Fanuc TP program (LS listing): SET_LOAD_PR.LS

/PROG  SET_LOAD_PR
/ATTR
OWNER		= MNEDITOR;
COMMENT		= "Set Grinder Load";
PROG_SIZE	= 3133;
CREATE		= DATE 28-11-03  TIME 05:11:18;
MODIFIED	= DATE 31-06-20  TIME 05:46:50;
FILE_NAME	= SET_SLOT;
VERSION		= 0;
LINE_COUNT	= 179;
MEMORY_SIZE	= 3693;
PROTECT		= READ_WRITE;
TCD:  STACK_SIZE	= 0,
      TASK_PRIORITY	= 50,
      TIME_SLICE	= 0,
      BUSY_LAMP_OFF	= 0,
      ABORT_REQUEST	= 0,
      PAUSE_REQUEST	= 0;
DEFAULT_GROUP	= *,*,*,*,*;
CONTROL_CODE	= 00000000 00000000;
/APPL
/APPL

AUTO_SINGULARITY_HEADER;
  ENABLE_SINGULARITY_AVOIDANCE   : TRUE;
/MN
   1:  JMP LBL[1] ;
   2:  !******************************* ;
   3:  !COMPANY ;
   4:  !PROJECT 0000000 ;
   5:  !CUSTOMER Example Cell ;
   6:  ! ;
   7:  !Date: March 24, 2022 ;
   8:  ! ;
   9:  !This program calculates the part ;
  10:  !tray LD position offsets. ;
  11:  ! ;
  12:  !******************************* ;
  13:  LBL[1:Begin] ;
  14:  !******************************* ;
  15:   ;
  16:  R[51:Part Style]=GI[3:Style Code]    ;
  17:   ;
  18:  !******************************* ;
  19:  LBL[5:Set Z values] ;
  20:  !******************************* ;
  21:   ;
  22:  SELECT R[51:Part Style]=1,JMP LBL[101] ;
  23:         =2,JMP LBL[102] ;
  24:         =3,JMP LBL[103] ;
  25:         =4,JMP LBL[104] ;
  26:         =5,JMP LBL[105] ;
  27:         =6,JMP LBL[106] ;
  28:         =7,JMP LBL[107] ;
  29:         =8,JMP LBL[108] ;
  30:         =9,JMP LBL[109] ;
  31:         =10,JMP LBL[110] ;
  32:         =11,JMP LBL[111] ;
  33:         =12,JMP LBL[112] ;
  34:         =13,JMP LBL[113] ;
  35:         =14,JMP LBL[114] ;
  36:         =15,JMP LBL[115] ;
  37:         =16,JMP LBL[116] ;
  38:         =17,JMP LBL[117] ;
  39:         =18,JMP LBL[118] ;
  40:         =19,JMP LBL[119] ;
  41:         =20,JMP LBL[120] ;
  42:         =21,JMP LBL[121] ;
  43:         =22,JMP LBL[122] ;
  44:         ELSE,JMP LBL[900] ;
  45:   ;
  46:  LBL[101] ;
  47:  R[56:Grinder Ld PR]=121    ;
  48:  R[57:Grinder Unld PR]=131    ;
  49:  R[58:Audit Ld PR]=151    ;
  50:  JMP LBL[200] ;
  51:   ;
  52:  LBL[102] ;
  53:  R[56:Grinder Ld PR]=122    ;
  54:  R[57:Grinder Unld PR]=132    ;
  55:  R[58:Audit Ld PR]=152    ;
  56:  JMP LBL[200] ;
  57:   ;
  58:  LBL[103] ;
  59:  R[56:Grinder Ld PR]=123    ;
  60:  R[57:Grinder Unld PR]=133    ;
  61:  R[58:Audit Ld PR]=153    ;
  62:  JMP LBL[200] ;
  63:   ;
  64:  LBL[104] ;
  65:  R[56:Grinder Ld PR]=124    ;
  66:  R[57:Grinder Unld PR]=134    ;
  67:  R[58:Audit Ld PR]=154    ;
  68:  JMP LBL[200] ;
  69:   ;
  70:  LBL[105] ;
  71:  R[56:Grinder Ld PR]=125    ;
  72:  R[57:Grinder Unld PR]=135    ;
  73:  R[58:Audit Ld PR]=155    ;
  74:  JMP LBL[200] ;
  75:   ;
  76:  LBL[106] ;
  77:  R[56:Grinder Ld PR]=126    ;
  78:  R[57:Grinder Unld PR]=136    ;
  79:  R[58:Audit Ld PR]=156    ;
  80:  JMP LBL[200] ;
  81:   ;
  82:  LBL[107] ;
  83:  R[56:Grinder Ld PR]=127    ;
  84:  R[57:Grinder Unld PR]=137    ;
  85:  R[58:Audit Ld PR]=157    ;
  86:  JMP LBL[200] ;
  87:   ;
  88:  LBL[108] ;
  89:  R[56:Grinder Ld PR]=128    ;
  90:  R[57:Grinder Unld PR]=138    ;
  91:  R[58:Audit Ld PR]=158    ;
  92:  JMP LBL[200] ;
  93:   ;
  94:  LBL[109] ;
  95:  R[56:Grinder Ld PR]=129    ;
  96:  R[57:Grinder Unld PR]=139    ;
  97:  R[58:Audit Ld PR]=159    ;
  98:  JMP LBL[200] ;
  99:   ;
 100:  LBL[110] ;
 101:  R[56:Grinder Ld PR]=130    ;
 102:  R[57:Grinder Unld PR]=140    ;
 103:  R[58:Audit Ld PR]=160    ;
 104:  JMP LBL[200] ;
 105:   ;
 106:  LBL[111] ;
 107:  R[56:Grinder Ld PR]=201    ;
 108:  R[57:Grinder Unld PR]=141    ;
 109:  JMP LBL[200] ;
 110:   ;
 111:  LBL[112] ;
 112:  R[56:Grinder Ld PR]=202    ;
 113:  R[57:Grinder Unld PR]=142    ;
 114:  JMP LBL[200] ;
 115:   ;
 116:  LBL[113] ;
 117:  R[56:Grinder Ld PR]=203    ;
 118:  R[57:Grinder Unld PR]=143    ;
 119:  JMP LBL[200] ;
 120:   ;
 121:  LBL[114] ;
 122:  R[56:Grinder Ld PR]=204    ;
 123:  R[57:Grinder Unld PR]=144    ;
 124:  JMP LBL[200] ;
 125:   ;
 126:  LBL[115] ;
 127:  R[56:Grinder Ld PR]=205    ;
 128:  R[57:Grinder Unld PR]=145    ;
 129:  JMP LBL[200] ;
 130:   ;
 131:  LBL[116] ;
 132:  R[56:Grinder Ld PR]=206    ;
 133:  R[57:Grinder Unld PR]=146    ;
 134:  JMP LBL[200] ;
 135:   ;
 136:  LBL[117] ;
 137:  R[56:Grinder Ld PR]=207    ;
 138:  R[57:Grinder Unld PR]=147    ;
 139:  JMP LBL[200] ;
 140:   ;
 141:  LBL[118] ;
 142:  R[56:Grinder Ld PR]=208    ;
 143:  R[57:Grinder Unld PR]=148    ;
 144:  JMP LBL[200] ;
 145:   ;
 146:  LBL[119] ;
 147:  R[56:Grinder Ld PR]=209    ;
 148:  R[57:Grinder Unld PR]=149    ;
 149:  JMP LBL[200] ;
 150:   ;
 151:  LBL[120] ;
 152:  R[56:Grinder Ld PR]=210    ;
 153:  R[57:Grinder Unld PR]=150    ;
 154:  JMP LBL[200] ;
 155:   ;
 156:  LBL[121] ;
 157:  R[56:Grinder Ld PR]=211    ;
 158:  R[57:Grinder Unld PR]=151    ;
 159:  JMP LBL[200] ;
 160:   ;
 161:  LBL[122] ;
 162:  R[56:Grinder Ld PR]=212    ;
 163:  R[57:Grinder Unld PR]=152    ;
 164:  JMP LBL[200] ;
 165:   ;
 166:   ;
 167:  !******************************* ;
 168:  LBL[200:End] ;
 169:  !******************************* ;
 170:  END ;
 171:   ;
 172:  !******************************* ;
 173:  LBL[900:Invalid Slot] ;
 174:  !******************************* ;
 175:   ;
 176:  GO[2:Application Fault]=10 ;
 177:  PAUSE ;
 178:  JMP LBL[1] ;
 179:   ;
/POS
/END
